FUNCTION_BLOCK CollectionDisposedEventHandler EXTENDS CollectionEventHandler

METHOD PUBLIC HandleEvent
VAR_INPUT
	Event : I_Event;
END_VAR
VAR
	disposedEvent : I_CollectionDisposedEvent;
END_VAR
IF __QUERYINTERFACE(Event, disposedEvent) THEN
	_eventReceived := TRUE;
	fromExpected := disposedEvent.Target = expectedOriginator;
END_IF
END_METHOD

END_FUNCTION_BLOCK

(* stored: Version 1.1.0.1, ProductVersion 3.1.4024.12
   POU CollectionDisposedEventHandler: Id {09cbe91e-c205-023a-23fe-74d36bd5bf22}, SpecialFunc None
   Method HandleEvent: Id {24998de9-ec1b-02b8-2176-477628cb27c5} *)
